TYPE typeMotionRowIO :
STRUCT
	
	//structure for a conventional motion (air cylinder, etc)

	iAdvanceDepth		AT %I* :BOOL;
	iReturnedDepth		AT %I* :BOOL;
	
	qAdvanceCoil		AT %Q* :BOOL;
	qReturnedCoil		AT %Q* :BOOL;
	

END_STRUCT
END_TYPE

(* stored: Version 1.1.0.1, ProductVersion 3.1.4024.12
   DUT typeMotionRowIO: Id {281ab22a-7d40-4753-af27-26dda4c2e6f0} *)
